// SIMATIC S7-200 project (STEP 7-Micro/WIN), CPU 221 REL 01.10

SYMBOL_TABLE USER1
dong_co_3        Q0.2
dong_co_2        Q0.1
dong_co_1        Q0.0
trung_gian_4     M0.4
trung_gian_3     M0.3
trung_gian_2     M0.2
trung_gian_1     M0.1
che_do_2         I0.2
che_do_1         I0.1
trung_gian       M0.0
s_top            I0.3
start            I0.0
END_SYMBOL_TABLE

ORGANIZATION_BLOCK MAIN:OB1
TITLE=PROGRAM COMMENTS
BEGIN
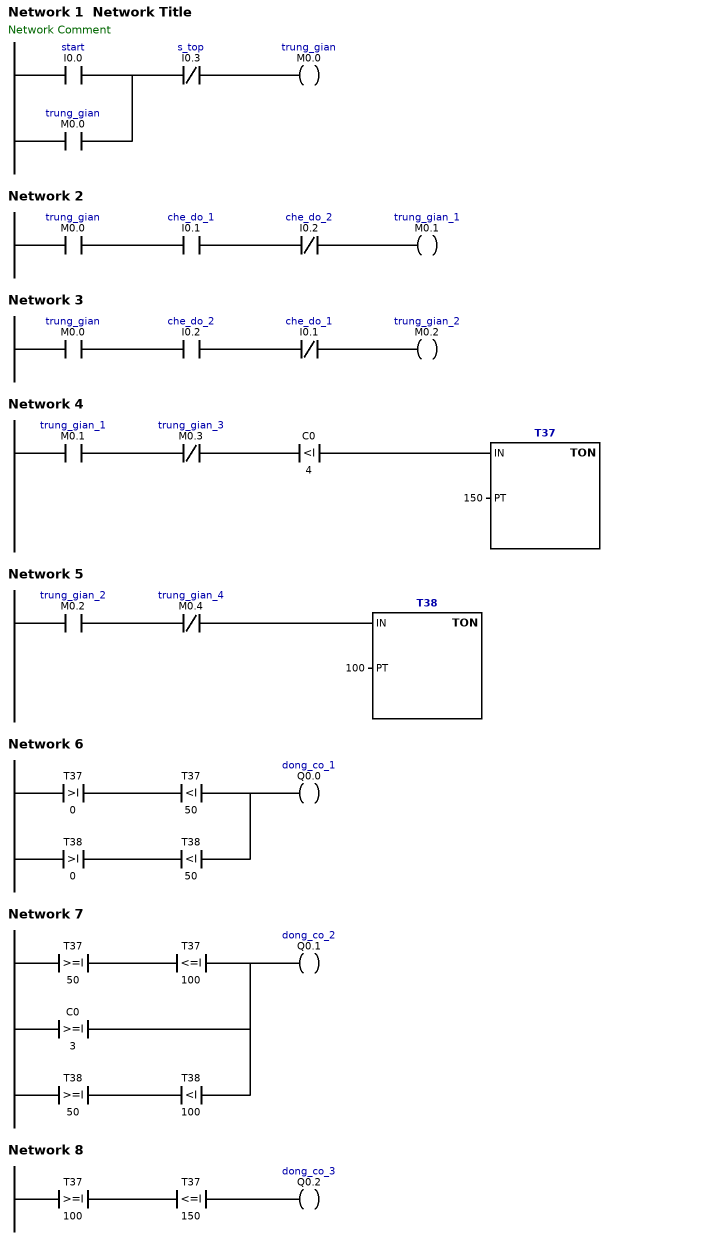
Network 1 // Network Title
// Network Comment
LD     start:I0.0
O      trung_gian:M0.0
AN     s_top:I0.3
=      trung_gian:M0.0
Network 2
LD     trung_gian:M0.0
A      che_do_1:I0.1
AN     che_do_2:I0.2
=      trung_gian_1:M0.1
Network 3
LD     trung_gian:M0.0
A      che_do_2:I0.2
AN     che_do_1:I0.1
=      trung_gian_2:M0.2
Network 4
LD     trung_gian_1:M0.1
AN     trung_gian_3:M0.3
AW<    C0, 4
TON    T37, 150
Network 5
LD     trung_gian_2:M0.2
AN     trung_gian_4:M0.4
TON    T38, 100
Network 6
LDW>   T37, 0
AW<    T37, 50
LDW>   T38, 0
AW<    T38, 50
OLD
=      dong_co_1:Q0.0
Network 7
LDW>=  T37, 50
AW<=   T37, 100
OW>=   C0, 3
LDW>=  T38, 50
AW<    T38, 100
OLD
=      dong_co_2:Q0.1
Network 8
LDW>=  T37, 100
AW<=   T37, 150
=      dong_co_3:Q0.2
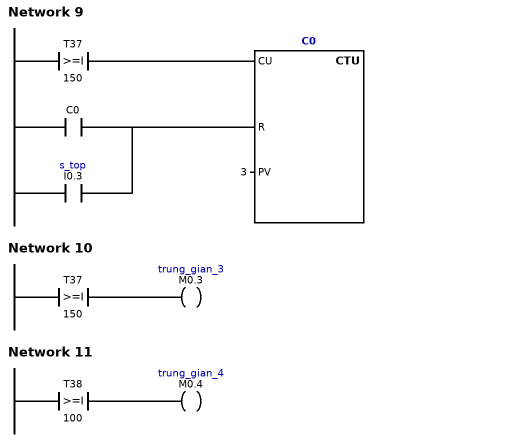
Network 9
LDW>=  T37, 150
LD     C0
O      s_top:I0.3
CTU    C0, 3
Network 10
LDW>=  T37, 150
=      trung_gian_3:M0.3
Network 11
LDW>=  T38, 100
=      trung_gian_4:M0.4
END_ORGANIZATION_BLOCK
